// TIA Portal V19 export
DATA_BLOCK "MappedCanProcessImageInputs"   // DB9
{ S7_Optimized_Access := 'FALSE' }
   VAR RETAIN
      statCanProcessImageInputs { S7_SetPoint := 'True'} : "typeCanProcessImageInputs";
   END_VAR
BEGIN
END_DATA_BLOCK
